FUNCTION_BLOCK StackMagazineController (* Basic Function Block Type *)
  (* Standard: 61499-2 *)
  (* Version 0.0, 2/16/2024, midxav, Template *)
  PACKAGE Main;
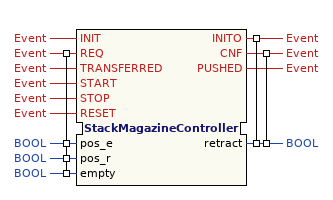
  EVENT_INPUT
    INIT; (* Initialization Request *)
    REQ WITH pos_e, pos_r, empty; (* Normal Execution Request *)
    TRANSFERRED;
    START;
    STOP;
    RESET;
  END_EVENT
  EVENT_OUTPUT
    INITO WITH retract; (* Initialization Confirm *)
    CNF WITH retract; (* Execution Confirmation *)
    PUSHED;
  END_EVENT
  VAR_INPUT
    pos_e : BOOL; (* Input event qualifier *)
    pos_r : BOOL;
    empty : BOOL;
  END_VAR
  VAR_OUTPUT
    retract : BOOL; (* Output event qualifier *)
  END_VAR
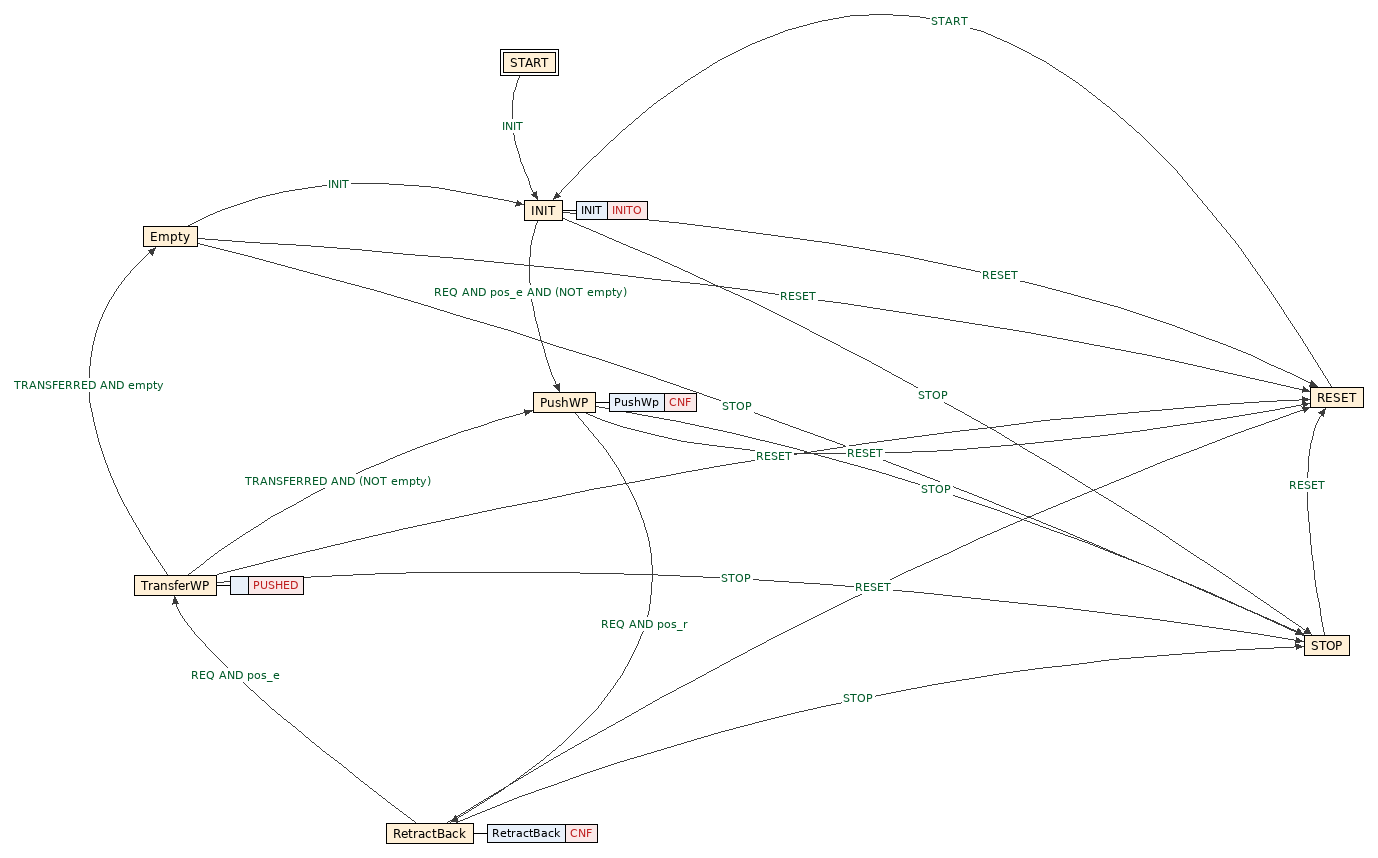
  EC_STATES
    START; (* Initial State *)
    INIT : INIT -> INITO; (* Initialization *)
    PushWP : PushWp -> CNF;
    RetractBack : RetractBack -> CNF;
    TransferWP : -> PUSHED;
    Empty;
    RESET;
    STOP;
  END_STATES
  EC_TRANSITIONS
    START TO INIT := INIT;
    INIT TO PushWP := REQ AND pos_e AND (NOT empty);
    PushWP TO RetractBack := REQ AND pos_r;
    RetractBack TO TransferWP := REQ AND pos_e;
    TransferWP TO PushWP := TRANSFERRED AND (NOT empty);
    TransferWP TO Empty := TRANSFERRED AND empty;
    Empty TO INIT := INIT;
    Empty TO RESET := RESET;
    TransferWP TO RESET := RESET;
    RetractBack TO RESET := RESET;
    PushWP TO RESET := RESET;
    INIT TO RESET := RESET;
    RESET TO INIT := START;
    INIT TO STOP := STOP;
    PushWP TO STOP := STOP;
    RetractBack TO STOP := STOP;
    TransferWP TO STOP := STOP;
    Empty TO STOP := STOP;
    STOP TO RESET := RESET;
  END_TRANSITIONS
  ALGORITHM INIT IN ST: (* Initialization algorithm *)
retract := FALSE;
  END_ALGORITHM
  ALGORITHM PushWp IN ST:
retract := TRUE;
  END_ALGORITHM
  ALGORITHM RetractBack IN ST:
retract := FALSE;
  END_ALGORITHM
END_FUNCTION_BLOCK
